// TIA Portal V18 export
// export: Created 2026-06-09T02:47:52.3796852Z, ExportSetting WithDefaults, DisplayName Totally Integrated Automation Portal, DisplayVersion V18, DisplayName TIA Portal Openness, DisplayVersion V18, DisplayName TIA Portal Version Control Interface, DisplayVersion V18, DisplayName STEP 7 Professional, DisplayVersion V18, DisplayName STEP 7 Safety, DisplayVersion V18, DisplayName WinCC Professional, DisplayVersion V18
VAR_GLOBAL   // PLC tag table "Default tag table"
   System_Byte AT %MB1 : Byte;
   FirstScan AT %M1.0 : Bool;
   DiagStatusUpdate AT %M1.1 : Bool;
   AlwaysTRUE AT %M1.2 : Bool;
   AlwaysFALSE AT %M1.3 : Bool;
   Clock_Byte AT %MB0 : Byte;
   Clock_10Hz AT %M0.0 : Bool;
   Clock_5Hz AT %M0.1 : Bool;
   "Clock_2.5Hz" AT %M0.2 : Bool;
   Clock_2Hz AT %M0.3 : Bool;
   "Clock_1.25Hz" AT %M0.4 : Bool;
   Clock_1Hz AT %M0.5 : Bool;
   "Clock_0.625Hz" AT %M0.6 : Bool;
   "Clock_0.5Hz" AT %M0.7 : Bool;
   rozlaczenie_tasmy AT %M100.2 : Bool;
   reset_licznika AT %M100.3 : Bool;
   zatrzymanie_tasmy AT %M101.2 : Bool;
   ilosc_butelek AT %MW10 : Int;
   reset_licznika_zak AT %M101.3 : Bool;
   ilosc_butelek_zak AT %MW16 : Int;
   Wylacznik_bezpieczenstwa AT %M205.0 : Bool;
   "Wlacznik/Wylacznik_glowny" AT %M206.0 : Bool;
   start_przenosik AT %M204.0 : Bool;
   stop_przenosnik AT %M204.1 : Bool;
   przenosnik_tasmowy AT %Q1.4 : Bool;
   wylacznik_przenosnika_tasmowego AT %I1.4 : Bool;
   wylacznik_nalewarki AT %I1.5 : Bool;
   wylacznik_zakrecarki AT %I1.6 : Bool;
   wylacznik_etykieciarki AT %I1.7 : Bool;
   wylacznik_pakowanie AT %I2.0 : Bool;
   samopod_start_zak AT %M102.3 : Bool;
   samopod_start_nal AT %M100.4 : Bool;
   Wlacznik_500ml AT %M207.0 : Bool;
   silownik AT %Q1.5 : Bool;
   sygnalizator_dzwiekowy AT %Q2.2 : Bool;
   robot AT %Q2.3 : Bool;
   lampa_przenosnik AT %Q2.4 : Bool;
   licznik_etykiet AT %MW50 : Int;
   cz_poj_ety AT %M210.0 : Bool;
   reset_licznika_etyk AT %M211.0 : Bool;
   pamiec_smakow AT %M100.5 : Bool;
   smak_zatrzymaj AT %M212.2 : Bool;
   czas_nalewarka AT %MD300 : Time;
   czas_pakowanie AT %MD304 : Time;
   czas_zakrecarka AT %MD308 : Time;
   cz_butelek_pakowanie AT %M230.0 : Bool;
   Tag_1 AT %MW400 : Word;
   licznik_przenosnik AT %MW30 : Int;
   res_licz_przen AT %M350.0 : Bool;
   Tag_4 AT %MD32 : Time;
   Tag_5 AT %M500.0 : Bool;
   res_licz_nalew AT %M350.1 : Bool;
   licznik_nalewarak AT %MW34 : Int;
   Tag_2 AT %M350.2 : Bool;
   Tag_3 AT %MW38 : Word;
   czas_move AT %MD312 : DWord;
   czas_w_int AT %MD316 : UDInt;
   Tag_6 AT %M320.0 : Bool;
   Tag_7 AT %MD321 : Time;
   Tag_8 AT %MD325 : Time;
   Tag_9 AT %MD329 : DInt;
   Tag_10 AT %I90.0 : Bool;
END_VAR
